FUNCTION_BLOCK FB_DataService
VAR_INPUT
END_VAR
VAR_OUTPUT
END_VAR
VAR
	fbStartProcess : NT_StartProcess;

	m_sCommandLine : STRING;
	m_sNetIP : STRING;
	m_sWorkingdirektory : STRING;
	m_sPathOfApplication : STRING;
	m_bStart : BOOL;
	m_eState : DATA_SERVICE_STATE;
	m_sErrCode : STRING;
	m_iReturnValue : DINT;
END_VAR

fbStartProcess.NETID 		:= m_sNetIP; // IP Adresse des Rechners auf dem die Zwillinge liegen
fbStartProcess.COMNDLINE 	:= m_sCommandLine; // Hier muss die ZwillingsID/ ProjektID übertragen werden
fbStartProcess.DIRNAME 		:= m_sWorkingdirektory; // Dieser Verzeichnis ist  vermutlich immer c:\TEMP
fbStartProcess.PATHSTR 		:= m_sPathOfApplication; // Pfad direkt zur DataService.exe wobei sich diese aus dem Zell-Namen ergibt 


IF fbStartProcess.ERR THEN // Fehlerabrage bereits vor der Zustandsmaschine 
	m_eState := DATA_SERVICE_STATE.e_ERROR;
END_IF 


CASE m_eState OF 
	DATA_SERVICE_STATE.e_IDLE:
	
		IF  m_bStart = TRUE THEN
			fbStartProcess.START := TRUE;
			m_bStart := FALSE; //Nurpositive Flanke übergeben		
		END_IF
	
		IF fbStartProcess.BUSY = TRUE THEN // Wenn der Funktionsblock selber Busy meldet in den nächsten Zustand
			m_eState := DATA_SERVICE_STATE.e_BUSY;
			fbStartProcess.START := FALSE;  
		END_IF
		
	DATA_SERVICE_STATE.e_BUSY:
	
 		IF fbStartProcess.BUSY = FALSE THEN
			IF m_iReturnValue = 1 THEN // Übergabewert der DataService.exe
				m_iReturnValue := 0; // Zurücksetzen für den nächsten Durchlauf
				m_eState := DATA_SERVICE_STATE.e_FINISHED;
			END_IF
			IF m_iReturnValue = 2 THEN
				m_eState := DATA_SERVICE_STATE.e_ERROR; 					
			END_IF		
		END_IF 
		
	DATA_SERVICE_STATE.e_FINISHED: // Zustand erforderlich da somit ein Zyklus lang abgefragt werden kann ob der Ablauf erfolgreich war
			
 		
		
	DATA_SERVICE_STATE.e_ERROR:
	
		m_sErrCode := UDINT_TO_STRING (fbStartProcess.ERRID); // Der Fehler wird als ganzzahl in den String geschrieben 
	
ELSE // Sicherheit bei falschem Wert
		m_eState := DATA_SERVICE_STATE.e_ERROR;
		m_sErrCode := 'Falscher Wert DataService-Status nicht vorhanden';
		
END_CASE

// Aufruf des Funktionblocks NT_StartProcess
fbStartProcess();

METHOD GetErrorCode : STRING
VAR_INPUT
END_VAR

VAR
END_VAR
GetErrorCode :=m_sErrCode;
END_METHOD

METHOD IsBusy : BOOL
VAR_INPUT
END_VAR
IF m_eState = DATA_SERVICE_STATE.e_BUSY THEN
	IsBusy := TRUE;
END_IF
END_METHOD

METHOD IsError : BOOL
VAR_INPUT
END_VAR
IF m_eState = DATA_SERVICE_STATE.e_ERROR THEN
	IsError := TRUE;
END_IF
END_METHOD

METHOD IsFinished : BOOL
VAR_INPUT
END_VAR
IF m_eState = DATA_SERVICE_STATE.e_FINISHED THEN
	IsFinished := TRUE;
END_IF
END_METHOD

METHOD IsIdle : BOOL
VAR_INPUT
END_VAR
IF m_eState = DATA_SERVICE_STATE.e_IDLE THEN
	IsIdle := TRUE;
END_IF
END_METHOD

METHOD SetCommandLine : BOOL
VAR_INPUT
	sCommandLine : STRING;
END_VAR
m_sCommandLine := sCommandLine;
END_METHOD

METHOD SetIdle : BOOL
VAR_INPUT
END_VAR
m_eState := DATA_SERVICE_STATE.e_IDLE;
END_METHOD

METHOD SetNetIP : BOOL
VAR_INPUT
	sNetIP : STRING;
END_VAR
m_sNetIP := sNetIP;
END_METHOD

METHOD SetPathOfApplication : BOOL
VAR_INPUT
	sPathOfApplication :STRING;
END_VAR
 m_sPathOfApplication := sPathOfApplication;
END_METHOD

METHOD SetWorkingDirectory : BOOL
VAR_INPUT
	sWorkingdirektory : STRING;
END_VAR
m_sWorkingdirektory := sWorkingdirektory;
END_METHOD

METHOD StartDataService : BOOL
VAR_INPUT
END_VAR
m_bStart := TRUE;
StartDataService := TRUE;
END_METHOD

END_FUNCTION_BLOCK

(* stored: Version 1.1.0.1, ProductVersion 3.1.4024.0
   POU FB_DataService: Id {7e8c7b75-930e-47cc-9741-8b2e8f213749}, SpecialFunc None
   Method GetErrorCode: Id {32dcc857-6da7-41b4-a061-ae1c26dd0071}
   Method IsBusy: Id {2393e7c9-8adc-4e42-9d3d-a62314aeb5e4}
   Method IsError: Id {db3fc9e9-0319-4d61-b839-13587aa67717}
   Method IsFinished: Id {4289dd15-334f-4299-8d4c-4094b8c5462f}
   Method IsIdle: Id {eb877cda-8ffc-48c4-81aa-406ee9d08783}
   Method SetCommandLine: Id {135f20ab-ff9a-44a5-888e-47e704a05b38}
   Method SetIdle: Id {71e274e4-7e13-4f34-94ae-c2c0ef0ff3df}
   Method SetNetIP: Id {ba7870e6-98f7-434a-80b3-5691cb675d7f}
   Method SetPathOfApplication: Id {cc576291-56f3-42b3-bdb1-334ae77c0e1c}
   Method SetWorkingDirectory: Id {2d36a123-4b31-42ed-abad-b3e4e179b4ac}
   Method StartDataService: Id {d2b001dd-860d-45df-89b6-51388711609b} *)
